PROGRAM MAIN
VAR
END_VAR

END_PROGRAM

(* stored: Version 1.1.0.1
   POU MAIN: Id {d214a1e0-6723-418d-953f-6111f09ba6c5} *)
